PROGRAM MAIN
VAR
	AmrModule	   : AmrModule('AMR Module');
	MachineHmiTree : GetSystemTreeJsonHmiVisitor<1000>('MAIN');
END_VAR

IF NOT AmrModule.Initialized THEN
	AmrModule.Initialize();
	MachineHmiTree.GetTree(AmrModule);
	RETURN;
END_IF

AmrModule.CyclicLogic();

END_PROGRAM

(* stored: Version 1.1.0.1
   POU MAIN: Id {967e055d-0eb5-42dc-b18d-7f8d4f634f3d}, SpecialFunc None *)
